Staubli VAL3: regular_place.pgx

program regular_place(tool x_tTool, mdesc x_mMdesc, mdesc x_mMdesc_slow, point x_pPoint_place, bool x_bBool_press, dio x_dDio_cy, bool x_bBool_bk)
  local point l_pPoint_drop
  local point l_pPoint_safe
  local point l_pPoint_press
  local point l_pPoint_aprch
begin
  //vertical regular drop process

  //----------------------------
  //control point preparation
  //----------------------------
  l_pPoint_safe=x_pPoint_place
  l_pPoint_safe.trsf.z=l_pPoint_safe.trsf.z+nNum_safe_h
  //----------------------------
  //approach point preparation
  //----------------------------
  l_pPoint_aprch=x_pPoint_place
  l_pPoint_aprch.trsf.z=l_pPoint_aprch.trsf.z+nNum_apporach_h
  //----------------------------
  //place point preparation
  //----------------------------
  l_pPoint_drop=x_pPoint_place

  l_pPoint_press = x_pPoint_place
  l_pPoint_press.trsf.z = l_pPoint_press.trsf.z-nNum_press

  ////to place via safe
  movej(l_pPoint_safe,x_tTool,x_mMdesc)
  waitEndMove()

  //corresponding cylinder extend
  if ioStatus(x_dDio_cy) >= 0
    //once io is working , on
    x_dDio_cy = true
    delay(nNum_cy_delay)
  endIf

  //---------------------------------
  // vertical should be linear mode
  // (Fast approach
  //---------------------------------
  movel(l_pPoint_aprch,x_tTool,x_mMdesc)
  waitEndMove()
  //---------------------------------
  // vertical should be linear mode
  //---------------------------------
  movel(l_pPoint_drop,x_tTool,x_mMdesc_slow)
  waitEndMove()
  //vg off
  if ioStatus(x_tTool.gripper) >= 0
    //once io is working
    close(x_tTool)
  endIf

  //additional press
  if x_bBool_press
    //---------------------------------
    // vertical should be linear mode
    //---------------------------------
    movel(l_pPoint_press,x_tTool,x_mMdesc)
    waitEndMove()
  endIf

  //additional back secure
  if ioStatus(dDio_bk) >= 0
    //once io is working and require back secure, on
    dDio_bk = x_bBool_bk
  endIf

  //----------
  //to safe
  // (Slow up
  //----------
  movel(l_pPoint_aprch,x_tTool,x_mMdesc_slow)
  waitEndMove()
  //---------------------------------
  // vertical should be linear mode
  //---------------------------------
  //to safe
  movel(l_pPoint_safe,x_tTool,x_mMdesc)
  waitEndMove()

  //corresponding cylinder extract
  if ioStatus(x_dDio_cy) >= 0
    //once io is working , off
    x_dDio_cy = false
  endIf

end
